FUNCTION_BLOCK CFB_FORECASTER (* Facade for PVForecaster and LoadForecaster to simplify interface *)
  (* Standard: 61499-2; Description: Function block for photovoltaic (PV) and load forecast generation. Outputs the difference between Ppv and Pload in W (positive = PV surplus, negative = PV deficit) along with an FCNF event every 15 min. An UDCNF event is output every min. IEC 61499 implementation of the "PVprog" algorithm. Original version's MIT license: Copyright (c) 2016 Joseph Bergner, Johannes Weniger, Tjarko Tjaden Permission is hereby granted, free of charge, to any person obtaining a copy of this software and associated documentation files (the "Software"), to deal in the Software without restriction, including without limitation the rights to use, copy, modify, merge, publish, distribute, sublicense, and/or sell copies of the Software, and to permit persons to whom the Software is furnished to do so, subject to the following conditions: The above copyright notice and this permission notice shall be included in all copies or substantial portions of the Software. THE SOFTWARE IS PROVIDED "AS IS", WITHOUT WARRANTY OF ANY KIND, EXPRESS OR IMPLIED, INCLUDING BUT NOT LIMITED TO THE WARRANTIES OF MERCHANTABILITY, FITNESS FOR A PARTICULAR PURPOSE AND NONINFRINGEMENT. IN NO EVENT SHALL THE AUTHORS OR COPYRIGHT HOLDERS BE LIABLE FOR ANY CLAIM, DAMAGES OR OTHER LIABILITY, WHETHER IN AN ACTION OF CONTRACT, TORT OR OTHERWISE, ARISING FROM, OUT OF OR IN CONNECTION WITH THE SOFTWARE OR THE USE OR OTHER DEALINGS IN THE SOFTWARE. *)
  (* Version 0.0, 2017-05-17, Marc Jakobi, HTW Berlin *)
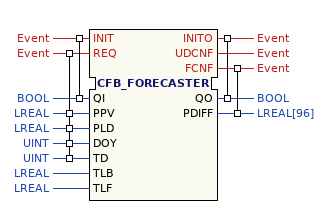
  EVENT_INPUT
    INIT WITH QI; (* Initialization Request *)
    REQ WITH PPV, PLD, DOY, TD; (* Normal Execution Request *)
  END_EVENT
  EVENT_OUTPUT
    INITO WITH QO; (* Initialization Confirm *)
    UDCNF; (* Update Execution Confirmation *)
    FCNF WITH PDIFF; (* Forecast Generation Confirmation (occurs every 15 min) *)
  END_EVENT
  VAR_INPUT
    QI : BOOL; (* Input event qualifier *)
    PPV : LREAL := 0; (* PV power in W *)
    PLD : LREAL := 0; (* Load in W *)
    DOY : UINT := 1; (* Day of the year [1..365] *)
    TD : UINT := 0; (* Time of day [min] [0..1439] *)
    TLB : LREAL := 3; (* Time frame to look back when generating PV power forecasts in h *)
    TLF : LREAL := 15; (* Time frame to forecast ahead (look forward) in h *)
  END_VAR
  VAR_OUTPUT
    QO : BOOL; (* Output event qualifier *)
    PDIFF : ARRAY [0..95] OF LREAL := 0; (* Power difference forecast in W (negative = PV deficit, positive = PV surplus) *)
  END_VAR
  FBS
    PVForecaster : PVForecaster;
    LoadForecaster : LoadForecaster;
    P_DIFF : FB_SUB_LREAL_ARR96;
    FREQ_SPLIT : E_SPLIT;
    UD_SPLIT2 : E_SPLIT;
    FCNF_REND : E_REND;
    UDCNF_REND : E_REND;
    FB_FORECAST_TIMER : FB_FORECAST_TIMER(RS := 15);
    UDCNF_SPLIT : E_SPLIT;
  END_FBS
  EVENT_CONNECTIONS
    PVForecaster.INITO TO LoadForecaster.INIT;
    LoadForecaster.INITO TO INITO;
    P_DIFF.CNF TO FCNF;
    FREQ_SPLIT.EO1 TO PVForecaster.FREQ;
    FREQ_SPLIT.EO2 TO LoadForecaster.FREQ;
    UD_SPLIT2.EO1 TO PVForecaster.UD;
    UD_SPLIT2.EO2 TO LoadForecaster.UD;
    PVForecaster.FCNF TO FCNF_REND.EI1;
    LoadForecaster.FCNF TO FCNF_REND.EI2;
    FCNF_REND.EO TO P_DIFF.REQ;
    PVForecaster.UDCNF TO UDCNF_REND.EI1;
    LoadForecaster.UDCNF TO UDCNF_REND.EI2;
    INIT TO FB_FORECAST_TIMER.INIT;
    FB_FORECAST_TIMER.INITO TO PVForecaster.INIT;
    FB_FORECAST_TIMER.FREQ TO FREQ_SPLIT.EI;
    FB_FORECAST_TIMER.UD TO UD_SPLIT2.EI;
    REQ TO FB_FORECAST_TIMER.REQ;
    UDCNF_SPLIT.EO2 TO FB_FORECAST_TIMER.UDCNF;
    UDCNF_SPLIT.EO1 TO UDCNF;
    UDCNF_REND.EO TO UDCNF_SPLIT.EI;
  END_CONNECTIONS
  DATA_CONNECTIONS
    PVForecaster.QO TO LoadForecaster.QI;
    PVForecaster.PF TO P_DIFF.IN1;
    LoadForecaster.PF TO P_DIFF.IN2;
    PPV TO PVForecaster.P;
    PLD TO LoadForecaster.P;
    TLB TO PVForecaster.TLB;
    LoadForecaster.QO TO QO;
    P_DIFF.OUT TO PDIFF;
    QI TO FB_FORECAST_TIMER.QI;
    DOY TO FB_FORECAST_TIMER.DOYIN;
    TD TO FB_FORECAST_TIMER.TDIN;
    FB_FORECAST_TIMER.QO TO PVForecaster.QI;
    FB_FORECAST_TIMER.DOYOUT TO PVForecaster.DOY;
    FB_FORECAST_TIMER.DOYOUT TO LoadForecaster.DOY;
    FB_FORECAST_TIMER.TDOUT TO LoadForecaster.TD;
    FB_FORECAST_TIMER.TDOUT TO PVForecaster.TD;
    TLF TO PVForecaster.TLF;
    TLF TO LoadForecaster.TLF;
  END_CONNECTIONS
END_FUNCTION_BLOCK
